TYPE
    CU00xComponents EXTENDS CUComponentsBase :
    STRUCT
        horizontalCylinder : TcoPneumatics.TcoCylinder(THISSTRUCT);
    END_STRUCT
END_TYPE

(* stored: Version 1.1.0.1, ProductVersion 3.1.4024.9
   DUT CU00xComponents: Id {4e1b0472-1d17-48ba-b026-d0be267cd4f2} *)
